FUNCTION_BLOCK INTERNAL fbDriveTest
VAR
	_drive : fbDrive;
END_VAR

_drive();

{attribute 'TcRpcEnable'}
METHOD INTERNAL MoveAbsoluteTest : BOOL
VAR_INPUT
	Position : LREAL;
	Speed : LREAL;
	AccDcc : LREAL;
END_VAR
MoveAbsoluteTest := _drive.MoveAbsolute(Position, 
										Speed, 
										AccDcc);
END_METHOD

END_FUNCTION_BLOCK

(* stored: Version 1.1.0.1, ProductVersion 3.1.4024.6
   POU fbDriveTest: Id {43a3ba59-a166-4056-ae4e-41b0b9ce866c}, SpecialFunc None
   Method MoveAbsoluteTest: Id {4400a0ac-b2f2-4507-bb4e-a4f15f1436cd} *)
